// TIA Portal V17 export
// export: Created 2024-09-02T12:49:57.0125926Z, ExportSetting WithDefaults, DisplayName Totally Integrated Automation Portal, DisplayVersion V17, DisplayName TIA Portal Openness, DisplayVersion V17, DisplayName TIA Portal Version Control Interface, DisplayVersion V17, DisplayName STEP 7 Professional, DisplayVersion V17, DisplayName STEP 7 Safety, DisplayVersion V17, DisplayName WinCC Professional, DisplayVersion V17
FUNCTION "SysFC_NumOfSQErrors" : Void   // FC126, LAD
TITLE = Count step errors / Schrittkettenfehler zaehlen
{ S7_Optimized_Access := 'TRUE' }
AUTHOR : OlegFuehrus
FAMILY : HMI
NAME : HMI
VERSION : 0.1
// stored: AutoNumber true, IsIECCheckEnabled false, SetENOAutomatically false, UDAEnableTagReadback false
   VAR_INPUT
      FLT : Bool;   // Schrittkettenfehler / Step sequence error
   END_VAR
   VAR_IN_OUT
      Fault_SQ : Bool;   // Meldung Fehler SK / Message Error SK
      NumOf_Fault_SQ : Int;   // Anzahl Fehler SK / Number of errors SK
   END_VAR
BEGIN

REGION Network 1: Count step errors / Schrittkettenfehler zaehlen
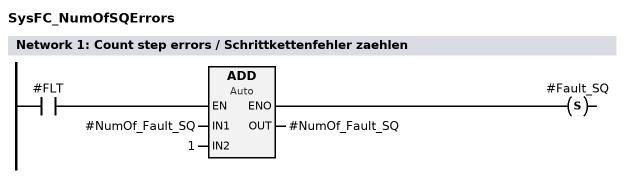
   RUNG wire#powerrail
      Contact( #FLT )
      Add(in1 := #NumOf_Fault_SQ, in2 := 1, out => #NumOf_Fault_SQ)
      S_Coil( #Fault_SQ )
   END_RUNG
   // the same network as SCL:
   IF #FLT THEN
       #NumOf_Fault_SQ := #NumOf_Fault_SQ + 1;
       #Fault_SQ := TRUE;
   END_IF;
END_REGION
END_FUNCTION
